// TwinCAT 3 PLC project PLC1
// ProgramVersion: 3.1.4024.0
// libraries:
//   Tc2_Standard, * (Beckhoff Automation GmbH)
//   Tc2_System, * (Beckhoff Automation GmbH)
//   Tc3_Module, * (Beckhoff Automation GmbH)
// project tree:
//   GVLs/ GVL_IO.TcGVL
//   / PlcTask.TcTTO
//   POUs/ MAIN.TcPOU
// real-time tasks:
//   TASK PlcTask: cycle T#10ms, priority 20, ADS port 350
// I/O:
//   DEVICE Device 3 (EtherCAT), AmsNetId 192.168.10.1.4.1
//     Term 11 (EK1100) [EK1100 EtherCAT Coupler (2A E-Bus)]
//       Term 12 (EL1012) [EL1012 2Ch. Dig. Input 24V, 10µs]
//       Term 13 (EL1012) [EL1012 2Ch. Dig. Input 24V, 10µs]
//       Term 14 (EL1012) [EL1012 2Ch. Dig. Input 24V, 10µs]
//       Term 15 (EL1012) [EL1012 2Ch. Dig. Input 24V, 10µs]
//       Term 16 (EL2004) [EL2004 4Ch. Dig. Output 24V, 0.5A]
//       Term 17 (EL4002) [EL4002 2Ch. Ana. Output 0-10V, 12bit]
//       Term 18 (EL9512) [EL9512 Power supply terminal 12V]
//       Term 19 (EL3102) [EL3102 2Ch. Ana. Input +/-10V, Diff.]
//       Term 26 (EL9011) [EL9011 End Terminal]
//     Term 20 (EK1100) [EK1100 EtherCAT Coupler (2A E-Bus)]
//       Term 21 (EL7211-0010) [EL7211-0010 1Ch. MDP742 Servo motor output stage with OCT (50V, 4.5A RMS)]
//       Term 22 (EL7211-0010) [EL7211-0010 1Ch. MDP742 Servo motor output stage with OCT (50V, 4.5A RMS)]
//       Term 23 (EL1904) [EL1904, 4 Ch. Safety Input 24V, TwinSAFE]
//         modules: Module 1 (FSOES)
//       Term 24 (EL2904) [EL2904, 4 Ch. Safety Output 24V, 0.5A, TwinSAFE]
//         modules: Module 1 (FSOES), Module 2 (DO)
//       Term 25 (EL6900) [EL6900, TwinSAFE PLC]
//       Term 27 (EL9011) [EL9011 End Terminal]
// variable links:
//   PLC1/PLC1 Instance <-> Device 3 (EtherCAT)/Term 11 (EK1100)/Term 12 (EL1012)
//     PlcTask Inputs/GVL_IO.bSwitchs[1] <-> Channel 1/Input
//     PlcTask Inputs/GVL_IO.bSwitchs[2] <-> Channel 2/Input
//   PLC1/PLC1 Instance <-> Device 3 (EtherCAT)/Term 11 (EK1100)/Term 13 (EL1012)
//     PlcTask Inputs/GVL_IO.bSwitchs[3] <-> Channel 1/Input
//     PlcTask Inputs/GVL_IO.bSwitchs[4] <-> Channel 2/Input
//   PLC1/PLC1 Instance <-> Device 3 (EtherCAT)/Term 11 (EK1100)/Term 14 (EL1012)
//     PlcTask Inputs/GVL_IO.bSwitchs[5] <-> Channel 1/Input
//     PlcTask Inputs/GVL_IO.bSwitchs[6] <-> Channel 2/Input
//   PLC1/PLC1 Instance <-> Device 3 (EtherCAT)/Term 11 (EK1100)/Term 15 (EL1012)
//     PlcTask Inputs/GVL_IO.bSwitchs[7] <-> Channel 1/Input
//     PlcTask Inputs/GVL_IO.bSwitchs[8] <-> Channel 2/Input
//   PLC1/PLC1 Instance <-> Device 3 (EtherCAT)/Term 11 (EK1100)/Term 16 (EL2004)
//     PlcTask Outputs/GVL_IO.bLamps[{1..4}] <-> Channel {1..4}/Output  (4 links)

CONFIGURATION PLC1
    RESOURCE PLC ON TwinCAT3
        TASK PlcTask(INTERVAL := T#10ms, PRIORITY := 20);
        PROGRAM MAIN WITH PlcTask : MAIN;
    END_RESOURCE
END_CONFIGURATION

// ---- GVLs/GVL_IO.TcGVL
{attribute 'qualified_only'}
VAR_GLOBAL
	bSwitchs AT%I* : ARRAY[1..8] OF BOOL;
	bLamps   AT%Q* : ARRAY[1..4] OF BOOL;

END_VAR

// ---- POUs/MAIN.TcPOU
PROGRAM MAIN
VAR
END_VAR

END_PROGRAM
